TYPE Terminal_Monitor_typ : 	
	STRUCT  
		SubSysName		: STRING[20];	
	END_STRUCT
END_TYPE

(* stored: Version 1.1.0.1, ProductVersion 3.1.4024.3
   DUT Terminal_Monitor_typ: Id {84b6a7fa-0044-09ee-350d-cce9e61d3d7e} *)
